(* IEC 61131-3 sources: Cybersecurity-projects-2024/openplc_logic/build, 2 files *)

(* ---- plc.st ---- *)
TYPE
  LOGLEVEL : (CRITICAL, WARNING, INFO, DEBUG) := INFO;
END_TYPE

FUNCTION_BLOCK LOGGER
  VAR_INPUT
    TRIG : BOOL;
    MSG : STRING;
    LEVEL : LOGLEVEL := INFO;
  END_VAR
  VAR
    TRIG0 : BOOL;
  END_VAR

  IF TRIG AND NOT TRIG0 THEN
  {{
   LogMessage(GetFbVar(LEVEL),(char*)GetFbVar(MSG, .body),GetFbVar(MSG, .len));
  }}
  END_IF;
  TRIG0:=TRIG;
END_FUNCTION_BLOCK

PROGRAM program0
  VAR
    sensor_0 : BOOL;
    sensor_1 : BOOL;
    arm_detect : BOOL;
    motor_0 : BOOL := True;
    motor_1 : BOOL := True;
    motor_2 : BOOL := True;
    motor_3 : BOOL := True;
    arm_Z : BOOL := False;
    arm_X : BOOL := False;
    arm_suck : BOOL := False;
  END_VAR
  VAR
    CL : INT := 0;
    TON0 : TON;
    TON1 : TON;
    TON2 : TON;
    TON3 : TON;
    TON4 : TON;
    TON5 : TON;
    TON6 : TON;
    _TMP_EQ40_OUT : BOOL;
    _TMP_AND97_OUT : BOOL;
    _TMP_ADD113_ENO : BOOL;
    _TMP_ADD113_OUT : INT;
    _TMP_EQ101_OUT : BOOL;
    _TMP_EQ9_ENO : BOOL;
    _TMP_EQ9_OUT : BOOL;
    _TMP_ADD5_ENO : BOOL;
    _TMP_ADD5_OUT : INT;
    _TMP_EQ12_OUT : BOOL;
    _TMP_EQ18_ENO : BOOL;
    _TMP_EQ18_OUT : BOOL;
    _TMP_ADD17_ENO : BOOL;
    _TMP_ADD17_OUT : INT;
    _TMP_EQ25_OUT : BOOL;
    _TMP_EQ31_ENO : BOOL;
    _TMP_EQ31_OUT : BOOL;
    _TMP_ADD30_ENO : BOOL;
    _TMP_ADD30_OUT : INT;
    _TMP_EQ43_OUT : BOOL;
    _TMP_EQ49_ENO : BOOL;
    _TMP_EQ49_OUT : BOOL;
    _TMP_ADD48_ENO : BOOL;
    _TMP_ADD48_OUT : INT;
    _TMP_EQ8_OUT : BOOL;
    _TMP_EQ63_ENO : BOOL;
    _TMP_EQ63_OUT : BOOL;
    _TMP_ADD62_ENO : BOOL;
    _TMP_ADD62_OUT : INT;
  END_VAR

  _TMP_EQ40_OUT := EQ(CL, 0);
  IF sensor_0 AND _TMP_EQ40_OUT THEN
    motor_0 := FALSE; (*reset*)
  END_IF;
  IF sensor_1 AND _TMP_EQ40_OUT THEN
    motor_1 := FALSE; (*reset*)
  END_IF;
  _TMP_AND97_OUT := AND(sensor_0 AND _TMP_EQ40_OUT, sensor_1 AND _TMP_EQ40_OUT);
  _TMP_ADD113_OUT := ADD(EN := _TMP_AND97_OUT, IN1 := 1, IN2 := 0, ENO => _TMP_ADD113_ENO);
  IF _TMP_ADD113_ENO THEN
      CL := _TMP_ADD113_OUT;
  END_IF;
  _TMP_EQ101_OUT := EQ(CL, 1);
  TON0(IN := arm_detect AND _TMP_EQ101_OUT, PT := T#1500ms);
  _TMP_EQ9_OUT := EQ(EN := TON0.Q, IN1 := CL, IN2 := 1, ENO => _TMP_EQ9_ENO);
  _TMP_ADD5_OUT := ADD(EN := _TMP_EQ9_OUT, IN1 := 2, ENO => _TMP_ADD5_ENO);
  IF _TMP_ADD5_ENO THEN
      CL := _TMP_ADD5_OUT;
  END_IF;
  IF _TMP_EQ101_OUT THEN
    arm_Z := TRUE; (*set*)
  END_IF;
  IF arm_detect AND _TMP_EQ101_OUT THEN
    arm_suck := TRUE; (*set*)
  END_IF;
  _TMP_EQ12_OUT := EQ(CL, 2);
  IF arm_detect AND _TMP_EQ12_OUT THEN
    arm_Z := FALSE; (*reset*)
  END_IF;
  TON1(IN := arm_detect AND _TMP_EQ12_OUT, PT := T#1500ms);
  _TMP_EQ18_OUT := EQ(EN := TON1.Q, IN1 := CL, IN2 := 2, ENO => _TMP_EQ18_ENO);
  _TMP_ADD17_OUT := ADD(EN := _TMP_EQ18_OUT, IN1 := 3, ENO => _TMP_ADD17_ENO);
  IF _TMP_ADD17_ENO THEN
      CL := _TMP_ADD17_OUT;
  END_IF;
  IF arm_detect AND _TMP_EQ12_OUT THEN
    arm_X := TRUE; (*set*)
  END_IF;
  _TMP_EQ25_OUT := EQ(CL, 3);
  IF arm_detect AND _TMP_EQ25_OUT THEN
    arm_Z := FALSE; (*reset*)
  END_IF;
  TON2(IN := arm_detect AND _TMP_EQ25_OUT, PT := T#1500ms);
  _TMP_EQ31_OUT := EQ(EN := TON2.Q, IN1 := CL, IN2 := 3, ENO => _TMP_EQ31_ENO);
  _TMP_ADD30_OUT := ADD(EN := _TMP_EQ31_OUT, IN1 := 4, ENO => _TMP_ADD30_ENO);
  IF _TMP_ADD30_ENO THEN
      CL := _TMP_ADD30_OUT;
  END_IF;
  IF arm_detect AND _TMP_EQ25_OUT THEN
    arm_X := TRUE; (*set*)
  END_IF;
  _TMP_EQ43_OUT := EQ(CL, 4);
  IF _TMP_EQ43_OUT THEN
    arm_Z := TRUE; (*set*)
  END_IF;
  IF _TMP_EQ43_OUT THEN
    arm_X := TRUE; (*set*)
  END_IF;
  TON3(IN := _TMP_EQ43_OUT, PT := T#2s);
  TON6(IN := TON3.Q, PT := T#200ms);
  _TMP_EQ49_OUT := EQ(EN := TON6.Q, IN1 := CL, IN2 := 4, ENO => _TMP_EQ49_ENO);
  _TMP_ADD48_OUT := ADD(EN := _TMP_EQ49_OUT, IN1 := 5, ENO => _TMP_ADD48_ENO);
  IF _TMP_ADD48_ENO THEN
      CL := _TMP_ADD48_OUT;
  END_IF;
  IF TON3.Q THEN
    arm_suck := FALSE; (*reset*)
  END_IF;
  _TMP_EQ8_OUT := EQ(CL, 5);
  IF _TMP_EQ8_OUT THEN
    arm_Z := FALSE; (*reset*)
  END_IF;
  IF _TMP_EQ8_OUT THEN
    arm_X := FALSE; (*reset*)
  END_IF;
  TON4(IN := _TMP_EQ8_OUT, PT := T#2s);
  TON5(IN := TON4.Q OR TON4.Q, PT := T#750ms);
  _TMP_EQ63_OUT := EQ(EN := TON5.Q, IN1 := CL, IN2 := 5, ENO => _TMP_EQ63_ENO);
  _TMP_ADD62_OUT := ADD(EN := _TMP_EQ63_OUT, IN1 := 0, ENO => _TMP_ADD62_ENO);
  IF _TMP_ADD62_ENO THEN
      CL := _TMP_ADD62_OUT;
  END_IF;
  IF sensor_0 AND _TMP_EQ40_OUT THEN
    motor_2 := FALSE; (*reset*)
  END_IF;
  IF sensor_1 AND _TMP_EQ40_OUT THEN
    motor_3 := FALSE; (*reset*)
  END_IF;
  IF TON4.Q THEN
    motor_0 := TRUE; (*set*)
  END_IF;
  IF TON4.Q THEN
    motor_2 := TRUE; (*set*)
  END_IF;
  IF TON4.Q THEN
    motor_1 := TRUE; (*set*)
  END_IF;
  IF TON4.Q THEN
    motor_3 := TRUE; (*set*)
  END_IF;
END_PROGRAM

CONFIGURATION Config0

  RESOURCE Res0 ON PLC
    TASK task0(INTERVAL := T#20ms,PRIORITY := 0);
    PROGRAM instance0 WITH task0 : program0;
  END_RESOURCE
END_CONFIGURATION

(* ---- generated_plc.st ---- *)
PROGRAM program0
  VAR
    sensor_0 AT %IX100.0 : BOOL;
    sensor_1 AT %IX100.1 : BOOL;
    arm_detect AT %IX100.2 : BOOL;
    motor_0 AT %QX100.0 : BOOL := True;
    motor_1 AT %QX100.1 : BOOL := True;
    motor_2 AT %QX100.2 : BOOL := True;
    motor_3 AT %QX100.3 : BOOL := True;
    arm_Z AT %QX100.4 : BOOL := False;
    arm_X AT %QX100.5 : BOOL := False;
    arm_suck AT %QX100.6 : BOOL := False;
  END_VAR
  VAR
    CL : INT := 0;
    TON0 : TON;
    TON1 : TON;
    TON2 : TON;
    TON3 : TON;
    TON4 : TON;
    TON5 : TON;
    TON6 : TON;
    _TMP_EQ40_OUT : BOOL;
    _TMP_AND97_OUT : BOOL;
    _TMP_ADD113_ENO : BOOL;
    _TMP_ADD113_OUT : INT;
    _TMP_EQ101_OUT : BOOL;
    _TMP_EQ9_ENO : BOOL;
    _TMP_EQ9_OUT : BOOL;
    _TMP_ADD5_ENO : BOOL;
    _TMP_ADD5_OUT : INT;
    _TMP_EQ12_OUT : BOOL;
    _TMP_EQ18_ENO : BOOL;
    _TMP_EQ18_OUT : BOOL;
    _TMP_ADD17_ENO : BOOL;
    _TMP_ADD17_OUT : INT;
    _TMP_EQ25_OUT : BOOL;
    _TMP_EQ31_ENO : BOOL;
    _TMP_EQ31_OUT : BOOL;
    _TMP_ADD30_ENO : BOOL;
    _TMP_ADD30_OUT : INT;
    _TMP_EQ43_OUT : BOOL;
    _TMP_EQ49_ENO : BOOL;
    _TMP_EQ49_OUT : BOOL;
    _TMP_ADD48_ENO : BOOL;
    _TMP_ADD48_OUT : INT;
    _TMP_EQ8_OUT : BOOL;
    _TMP_EQ63_ENO : BOOL;
    _TMP_EQ63_OUT : BOOL;
    _TMP_ADD62_ENO : BOOL;
    _TMP_ADD62_OUT : INT;
  END_VAR

  _TMP_EQ40_OUT := EQ(CL, 0);
  IF sensor_0 AND _TMP_EQ40_OUT THEN
    motor_0 := FALSE; (*reset*)
  END_IF;
  IF sensor_1 AND _TMP_EQ40_OUT THEN
    motor_1 := FALSE; (*reset*)
  END_IF;
  _TMP_AND97_OUT := AND(sensor_0 AND _TMP_EQ40_OUT, sensor_1 AND _TMP_EQ40_OUT);
  _TMP_ADD113_OUT := ADD(EN := _TMP_AND97_OUT, IN1 := 1, IN2 := 0, ENO => _TMP_ADD113_ENO);
  IF _TMP_ADD113_ENO THEN
      CL := _TMP_ADD113_OUT;
  END_IF;
  _TMP_EQ101_OUT := EQ(CL, 1);
  TON0(IN := arm_detect AND _TMP_EQ101_OUT, PT := T#1500ms);
  _TMP_EQ9_OUT := EQ(EN := TON0.Q, IN1 := CL, IN2 := 1, ENO => _TMP_EQ9_ENO);
  _TMP_ADD5_OUT := ADD(EN := _TMP_EQ9_OUT, IN1 := 2, ENO => _TMP_ADD5_ENO);
  IF _TMP_ADD5_ENO THEN
      CL := _TMP_ADD5_OUT;
  END_IF;
  IF _TMP_EQ101_OUT THEN
    arm_Z := TRUE; (*set*)
  END_IF;
  IF arm_detect AND _TMP_EQ101_OUT THEN
    arm_suck := TRUE; (*set*)
  END_IF;
  _TMP_EQ12_OUT := EQ(CL, 2);
  IF arm_detect AND _TMP_EQ12_OUT THEN
    arm_Z := FALSE; (*reset*)
  END_IF;
  TON1(IN := arm_detect AND _TMP_EQ12_OUT, PT := T#1500ms);
  _TMP_EQ18_OUT := EQ(EN := TON1.Q, IN1 := CL, IN2 := 2, ENO => _TMP_EQ18_ENO);
  _TMP_ADD17_OUT := ADD(EN := _TMP_EQ18_OUT, IN1 := 3, ENO => _TMP_ADD17_ENO);
  IF _TMP_ADD17_ENO THEN
      CL := _TMP_ADD17_OUT;
  END_IF;
  IF arm_detect AND _TMP_EQ12_OUT THEN
    arm_X := TRUE; (*set*)
  END_IF;
  _TMP_EQ25_OUT := EQ(CL, 3);
  IF arm_detect AND _TMP_EQ25_OUT THEN
    arm_Z := FALSE; (*reset*)
  END_IF;
  TON2(IN := arm_detect AND _TMP_EQ25_OUT, PT := T#1500ms);
  _TMP_EQ31_OUT := EQ(EN := TON2.Q, IN1 := CL, IN2 := 3, ENO => _TMP_EQ31_ENO);
  _TMP_ADD30_OUT := ADD(EN := _TMP_EQ31_OUT, IN1 := 4, ENO => _TMP_ADD30_ENO);
  IF _TMP_ADD30_ENO THEN
      CL := _TMP_ADD30_OUT;
  END_IF;
  IF arm_detect AND _TMP_EQ25_OUT THEN
    arm_X := TRUE; (*set*)
  END_IF;
  _TMP_EQ43_OUT := EQ(CL, 4);
  IF _TMP_EQ43_OUT THEN
    arm_Z := TRUE; (*set*)
  END_IF;
  IF _TMP_EQ43_OUT THEN
    arm_X := TRUE; (*set*)
  END_IF;
  TON3(IN := _TMP_EQ43_OUT, PT := T#2s);
  TON6(IN := TON3.Q, PT := T#200ms);
  _TMP_EQ49_OUT := EQ(EN := TON6.Q, IN1 := CL, IN2 := 4, ENO => _TMP_EQ49_ENO);
  _TMP_ADD48_OUT := ADD(EN := _TMP_EQ49_OUT, IN1 := 5, ENO => _TMP_ADD48_ENO);
  IF _TMP_ADD48_ENO THEN
      CL := _TMP_ADD48_OUT;
  END_IF;
  IF TON3.Q THEN
    arm_suck := FALSE; (*reset*)
  END_IF;
  _TMP_EQ8_OUT := EQ(CL, 5);
  IF _TMP_EQ8_OUT THEN
    arm_Z := FALSE; (*reset*)
  END_IF;
  IF _TMP_EQ8_OUT THEN
    arm_X := FALSE; (*reset*)
  END_IF;
  TON4(IN := _TMP_EQ8_OUT, PT := T#2s);
  TON5(IN := TON4.Q OR TON4.Q, PT := T#750ms);
  _TMP_EQ63_OUT := EQ(EN := TON5.Q, IN1 := CL, IN2 := 5, ENO => _TMP_EQ63_ENO);
  _TMP_ADD62_OUT := ADD(EN := _TMP_EQ63_OUT, IN1 := 0, ENO => _TMP_ADD62_ENO);
  IF _TMP_ADD62_ENO THEN
      CL := _TMP_ADD62_OUT;
  END_IF;
  IF sensor_0 AND _TMP_EQ40_OUT THEN
    motor_2 := FALSE; (*reset*)
  END_IF;
  IF sensor_1 AND _TMP_EQ40_OUT THEN
    motor_3 := FALSE; (*reset*)
  END_IF;
  IF TON4.Q THEN
    motor_0 := TRUE; (*set*)
  END_IF;
  IF TON4.Q THEN
    motor_2 := TRUE; (*set*)
  END_IF;
  IF TON4.Q THEN
    motor_1 := TRUE; (*set*)
  END_IF;
  IF TON4.Q THEN
    motor_3 := TRUE; (*set*)
  END_IF;
END_PROGRAM

CONFIGURATION Config0

  RESOURCE Res0 ON PLC
    TASK task0(INTERVAL := T#20ms,PRIORITY := 0);
    PROGRAM instance0 WITH task0 : program0;
  END_RESOURCE
END_CONFIGURATION
